//ABS(m_cmdJntPos[7]-curJntPos[7])> m_maxTrackErr OR
//Calculate the deviation of J4 from the zero point
m_instruZeroDeviationJ4:=m_PowerboxZeroPos[1,4] - i_slaveArm.linkSingle[4+3] ;
IF m_instruZeroDeviationJ4>2*PI THEN
	m_instruZeroDeviationJ4:=m_instruZeroDeviationJ4-2*PI;
END_IF

// traj plan
FOR i:=1 TO 5 DO
	m_jntOTG[i].run(m_targetMountPos[i+3],0.0, o_cmdAcc=>m_cmdJntAcc[3+i],o_cmdVel=>m_cmdJntVel[3+i],o_cmdPos=>m_cmdJntPos[i+3]);
END_FOR
END_METHOD

METHOD PUBLIC init : BOOL
VAR_IN_OUT CONSTANT
	i_slaveArm	:FB_SlaveArm;
END_VAR
VAR_IN_OUT 
	r_slaveArmCtrlCmd :ST_SlaveArmCtrlCmds;
END_VAR

VAR
	i : INT;
END_VAR
SUPER^.Init(i_slaveArm,r_slaveArmCtrlCmd);

// check if to hold the command joint position unchanged
checkToHoldLastCmds(i_slaveArm,r_slaveArmCtrlCmd);
FOR i:=1 TO 5 DO
	m_targetMountPos[i+3]:=m_cmdJntPos[i+3];
	m_jntOTG[i].init(m_targetMountPos[i+3], 0,m_instruMountVel, m_instruMountAcc, g_slaveArmCtrlCycleTime);
	m_jointMounted[i]:=FALSE;
END_FOR

m_mountStatus:=0;
// check instrument type to get mount joint index and zero position
IF i_slaveArm.instrument.InstruReadPara.m_Instrutype <> InstruType_UNKNOWM THEN
	m_jointMounted[5]:=TRUE;

END_IF


//Update the IP and port number of the operating arm
i_slaveArm.instrument.InstruReadPara.i_ArmNetId:=GVL_SlaveMotorParameters.g_slaveArmNetID[1];
i_slaveArm.instrument.InstruReadPara.i_JointInstruAddr:=GVL_SlaveMotorParameters.g_slaveJointNetPort[1,4];

m_Error:=FALSE;
m_ErrorID:=0;
END_METHOD

END_FUNCTION_BLOCK

// ---- FBs_SlaveControllers/FB_SlaveCtrlMasterSlave.TcPOU
// Brief: Slave Arm MasterSlave controller
FUNCTION_BLOCK PUBLIC FB_SlaveCtrlMasterSlave EXTENDS FB_SlaveArmCtrlBase
VAR_INPUT
END_VAR
VAR_OUTPUT
END_VAR
VAR
// ################ variables for single joint test ##################
	m_initJntPos :Vec8d;
	m_jntMotionFreq :Vec8d :=[0.1, 0.1, 0.1, 0, 0, 0, 0, 0];
	m_jntMotionRange :Vec8d :=[pi/6, pi/4, 0.1, 0, 0, 0, 0];
	testIdx :INT :=1;
	
//####################################################################

END_VAR

METHOD PROTECTED calcCmdJntPos : BOOL
VAR_INPUT
	motionScale :LREAL;
	masterIdx :INT;
END_VAR

VAR_IN_OUT CONSTANT
	i_slaveArm :FB_SlaveArm;
	i_masterStatus :ST_MasterStatus;
END_VAR
VAR 
	i:INT :=0;
	errThres :LREAL;
END_VAR
// Just for joint controller test
IF testIdx >0 THEN
	m_cmdJntPos[testIdx]:=m_initJntPos[testIdx]+m_jntMotionRange[testIdx]* SIN(2*pi*m_jntMotionFreq[testIdx]*m_timePeriod);
	m_cmdJntVel[testIdx]:=m_jntMotionRange[testIdx]*2*pi*m_jntMotionFreq[testIdx]*COS(2*pi*m_jntMotionFreq[testIdx]*m_timePeriod);
END_IF



FOR i:=1 TO 8 DO 
	IF i=3 THEN
		errThres := 0.01;
	ELSE
		errThres :=5*g_deg2rad;
	END_IF
	
	IF ABS(m_cmdJntPos[i]-i_slaveArm.curJntPos[i])>errThres THEN
		m_isFinished:=TRUE;
	END_IF
	
END_FOR
END_METHOD

// override this function in each exact controller
METHOD PROTECTED calcCmdJntTrq : BOOL
VAR_INPUT
	motionScale :LREAL;
	masterIdx :INT;
END_VAR

VAR_IN_OUT CONSTANT
	i_slaveArm :FB_SlaveArm;
	i_masterStatus :ST_MasterStatus;
END_VAR
VAR 
	nullspaceMat :Mat7d;
	ctrlTrq : Vec7d;
END_VAR
// set joint torque to zero in default
m_cmdJntTrq := g_zeroVec8d;
END_METHOD

METHOD PUBLIC init : BOOL
VAR_IN_OUT CONSTANT
	i_slaveArm	:FB_SlaveArm;
END_VAR
VAR_IN_OUT 
	r_slaveArmCtrlCmd :ST_SlaveArmCtrlCmds;
END_VAR
SUPER^.Init(i_slaveArm,r_slaveArmCtrlCmd);

m_jntOPMode := g_slaveAllPosTrqMode;

m_initJntPos :=i_slaveArm.curJntPos;
END_METHOD

END_FUNCTION_BLOCK

// ---- FBs_SlaveControllers/FB_SlaveCtrlScopeReady.TcPOU
// Brief:Scope Ready
FUNCTION_BLOCK PUBLIC FB_SlaveCtrlScopeReady EXTENDS FB_SlaveArmCtrlBase
VAR_INPUT
END_VAR
VAR_OUTPUT
END_VAR
VAR
END_VAR

METHOD PUBLIC init : BOOL
VAR_IN_OUT CONSTANT
	i_slaveArm	:FB_SlaveArm;
END_VAR
VAR_IN_OUT 
	r_slaveArmCtrlCmd :ST_SlaveArmCtrlCmds;
END_VAR


VAR
	j:INT;
	maxJntErr:LREAL;
	jntCtrlErr:Vec7d;
END_VAR
SUPER^.Init(i_slaveArm,r_slaveArmCtrlCmd);

// check if to hold the command joint position unchanged
checkToHoldLastCmds(i_slaveArm,r_slaveArmCtrlCmd);
END_METHOD

END_FUNCTION_BLOCK

// ---- FBs_SlaveControllers/FB_SlaveCtrlEndoscope.TcPOU
// Brief: Slave Arm Endoscope Control
FUNCTION_BLOCK PUBLIC FB_SlaveCtrlEndoscope EXTENDS FB_SlaveArmCtrlBase
VAR_INPUT
END_VAR
VAR_OUTPUT
END_VAR
VAR
END_VAR

END_FUNCTION_BLOCK

// ---- FBs_SlaveControllers/FB_SlaveCtrlAdjust.TcPOU
// Brief: Slave Arm Adjust
FUNCTION_BLOCK PUBLIC FB_SlaveCtrlAdjust EXTENDS FB_SlaveArmCtrlBase
VAR_INPUT
END_VAR
VAR_OUTPUT
END_VAR
VAR
END_VAR

METHOD PUBLIC init : BOOL
VAR_IN_OUT CONSTANT
	i_slaveArm	:FB_SlaveArm;
END_VAR
VAR_IN_OUT 
	r_slaveArmCtrlCmd :ST_SlaveArmCtrlCmds;
END_VAR
SUPER^.Init(i_slaveArm,r_slaveArmCtrlCmd);

// check if to hold the command joint position unchanged
checkToHoldLastCmds(i_slaveArm,r_slaveArmCtrlCmd);
END_METHOD

END_FUNCTION_BLOCK

// ---- FBs_SlaveControllers/FB_SlaveCtrlGraCali.TcPOU
// Brief: Slave Arm Gravity Calibration
FUNCTION_BLOCK PUBLIC FB_SlaveCtrlGraCali EXTENDS FB_SlaveArmCtrlBase
VAR_INPUT
END_VAR
VAR_OUTPUT
END_VAR
VAR
// cali trajectory
	m_caliMotionSegs :INT :=3;
	m_graCaliTraj:ARRAY [1..3, 1..g_sJntNum] OF LREAL:=
		[-pi/6, -PI/2+pi/6, 0.4, 	0, 0, 0, 0,0,
		 pi/6, 	-PI/2-pi/4, 0.2, 	0, 0, 0, 0,0,
		 -pi/6, -PI/2+pi/6, 0.4, 	0, 0, 0, 0,0];
		 
	m_caliMaxjntVel:Vec8d:=[8(0.02)];
	m_caliMaxjntAcc:Vec8d:=[8(0.5)];
	m_caliMaxjntJerk:Vec8d:=[8(2.0)];
	
	m_caliTrajIdx: INT := 1;
	m_caliPlanner: ARRAY[1..3] OF FB_TrajMoveJ;
	
END_VAR

// override this function in each exact controller
METHOD PROTECTED calcCmdJntPos : BOOL
VAR_INPUT
	motionScale :LREAL;
	masterIdx :INT;
END_VAR

VAR_IN_OUT CONSTANT
	i_slaveArm :FB_SlaveArm;
	i_masterStatus :ST_MasterStatus;
END_VAR

VAR 
	i :INT;
	curJntVel :Vec8d;
END_VAR
// check if planner is ready
IF m_caliPlanner[m_caliTrajIdx].isGene = FALSE THEN
	calcCmdJntPos:=FALSE;
	RETURN;
END_IF

// traj plan
calcCmdJntPos :=m_caliPlanner[m_caliTrajIdx].evaluate(m_timePeriod, jntPos=> m_cmdJntPos, jntVel=>m_cmdJntVel, jntAcc=> m_cmdJntAcc);

// check if to transit to next segment
curJntVel :=i_slaveArm.curJntVel;
IF(m_timePeriod > m_caliPlanner[m_caliTrajIdx].duration  AND vecNorm(curJntVel)<7*GVL_SlaveControlParameters.g_jntStaticVelThres) THEN
	m_caliTrajIdx:=m_caliTrajIdx+1;
	m_timePeriod:=0;
END_IF

// check if to terminated
IF(m_caliTrajIdx > m_caliMotionSegs) THEN
	m_isFinished:=TRUE;
END_IF
END_METHOD

METHOD PUBLIC init : BOOL
VAR_IN_OUT CONSTANT
	i_slaveArm	:FB_SlaveArm;
END_VAR
VAR_IN_OUT 
	r_slaveArmCtrlCmd :ST_SlaveArmCtrlCmds;
END_VAR

VAR
	i,j :INT;
	startJntPos,endJntPos :Vec8d;
END_VAR
SUPER^.Init(i_slaveArm,r_slaveArmCtrlCmd);
m_caliTrajIdx :=1;

// traj plan
// fisrt segment
startJntPos:=i_slaveArm.curJntPos;
FOR j:=1 TO g_sJntNum DO 
endJntPos[j]:=m_graCaliTraj[1,j];
END_FOR
m_caliPlanner[1].init(startJntPos,endJntPos,m_caliMaxjntVel, m_caliMaxJntAcc, m_caliMaxJntJerk);

// other segments
FOR i:=2 TO m_caliMotionSegs DO 
	FOR j:=1 TO g_sJntNum DO 
		startJntPos[j]:=m_graCaliTraj[i-1,j];
		endJntPos[j]:=m_graCaliTraj[i,j];
	END_FOR
	m_caliPlanner[i].init(startJntPos,endJntPos,m_caliMaxjntVel, m_caliMaxJntAcc, m_caliMaxJntJerk);
END_FOR
END_METHOD

END_FUNCTION_BLOCK

// ---- AgiMaths/deg2rad.TcPOU
FUNCTION deg2rad : lreal
VAR_INPUT
	angle_deg:lreal;
END_VAR
VAR
END_VAR

deg2rad:=angle_deg*pi/180;

END_FUNCTION

// ---- FBs_BasicControllers/FBMacroJntControl.TcPOU
// Author: Feijian Ni
// Date: 2023.11.22
FUNCTION_BLOCK FBMacroJntControl
VAR_INPUT
END_VAR
VAR_OUTPUT
END_VAR
VAR
	//TODO: move to GVLs 
	// control paramters
	m_macroJntKp:ARRAY[1..3] OF LREAL:=[1200,10,10];
	m_macroJntKd:ARRAY[1..4] OF LREAL:=[100,1.0,1.0];
	m_macroJntKi:ARRAY[1..4] OF LREAL:=[3000,0,0,0];
	m_macroJntKiLimit:ARRAY[1..4] OF LREAL:=[3(1500.0)];
	m_macroJnttrlLimit:ARRAY[1..4] OF LREAL:=[3(3500.0)];
	m_jntTargetPosLpfCutoffFreq:LREAL:=10;
	m_curJntVelLpfCutoffFreq:LREAL:=30;
	
	// filter for target joint position
	m_cmdPosLpf:ARRAY[1..3] OF FBLowPassFilter;
	
	// filter for current joint velocity
	m_curJntVelLpf:ARRAY[1..3] OF FBLowPassFilter;
	
	// max command joint velocity
	m_maxJntVel:ARRAY[1..3] OF LREAL:=[1.5, 0.1, 0.1];
	
	// arm index for grip control
	m_armIdx:INT;
	
	// final target macro joint position
	m_targetJntPos:ARRAY[1..3] OF LREAL;
	
	// position tracking error
	m_posErr:ARRAY[1..3] OF LREAL;
	
	// max position error for safety check
	m_safetyPosErr:ARRAY[1..3] OF LREAL:=[5.0*pi/180,5.0*pi/180,0.01];
	
	// command macro joint position and veloicty for next cycle
	m_cmdJntPos:ARRAY[1..3] OF LREAL;
	m_cmdJntVel:ARRAY[1..3] OF LREAL;

	// current  macro joint position and veloicty for next cycle
	m_curJntPos:ARRAY[1..3] OF LREAL;
	m_curJntVel:ARRAY[1..3] OF LREAL;
	
	// PID for joint position
	m_jntPIDCtrl:ARRAY[1..3] OF FBPID;
	m_jntCtrlTrq:ARRAY[1..3] OF LREAL;
	
END_VAR

METHOD init : BOOL
VAR_INPUT
	i_armIdx:INT;
END_VAR

VAR
	i,j:INT;
	currentRatioMotor2Jnt:LREAL;
END_VAR
m_armIdx:=i_armIdx;

// get current instrument orientation
m_curJntPos[1]:=Robot_Status.Robot_Current_DH_Joint_Position_M3[m_armIdx].q1;
m_curJntPos[2]:=Robot_Status.Robot_Current_DH_Joint_Position_M3[m_armIdx].q2;
m_curJntPos[3]:=Robot_Status.Robot_Current_DH_Joint_Position_M3[m_armIdx].q3;
FOR i:=1 TO 3  DO 
	m_targetJntPos[i]:=m_curJntPos[i];
	m_cmdJntPos[i]:=m_curJntPos[i];
	m_cmdJntVel[i]:=0;
	m_curJntVel[i]:=0;
END_FOR

// init controller
FOR i:=1 TO 3 DO
	currentRatioMotor2Jnt:=GVL_system_parameters.arm_joint_transmition_efficiency[i-1+Gvl_IO.Joint6]*GVL_system_parameters.arm_joint_torque_constant[i-1+Gvl_IO.Joint6]
							*GVL_system_parameters.transmission_ratio[m_armIdx, i-1+Gvl_IO.Joint6]/1000;
	m_jntPIDCtrl[i].init(GVL_system_parameters.cycle_robot,m_macroJntKp[i],m_macroJntKd[i],m_macroJntKi[i],
		m_macroJntKiLimit[i]* currentRatioMotor2Jnt,	m_macroJnttrlLimit[i]*currentRatioMotor2Jnt);
END_FOR

// init low pass filter
FOR i:=1 TO 3 DO
	m_cmdPosLpf[i].init(i_filterOrd:=1,i_cutoffFreq:=m_jntTargetPosLpfCutoffFreq,i_sampleFreq:=1000);
	m_curJntVelLpf[i].init(i_filterOrd:=1,i_cutoffFreq:=m_curJntVelLpfCutoffFreq,i_sampleFreq:=1000);
END_FOR
END_METHOD

METHOD run : BOOL
VAR_INPUT
	// target joint position in DH model 3
	i_targetJntPos:ARRAY[1..3] OF LREAL;

END_VAR

VAR_OUTPUT
	// motor control current
	o_cmdMotorTrq:ARRAY[1..3] OF LREAL;
END_VAR

VAR
	i: INT;
END_VAR
// fitl target joint position
FOR i:=1 TO 3 DO
	m_targetJntPos[i]:=m_cmdPosLpf[i].run(i_targetJntPos[i]);
END_FOR

// get current joint position
m_curJntPos[1]:=Robot_Status.Robot_Current_DH_Joint_Position_M3[m_armIdx].q1;
m_curJntPos[2]:=Robot_Status.Robot_Current_DH_Joint_Position_M3[m_armIdx].q2;
m_curJntPos[3]:=Robot_Status.Robot_Current_DH_Joint_Position_M3[m_armIdx].q3;

// get current joint velocity
m_curJntVel[1]:=m_curJntVelLpf[1].run(Robot_Status.Robot_Current_Joint_Velocity_V2[m_armIdx,6]);
m_curJntVel[2]:=m_curJntVelLpf[2].run(Robot_Status.Robot_Current_Joint_Velocity_V2[m_armIdx,10]);
m_curJntVel[3]:=m_curJntVelLpf[3].run(Robot_Status.Robot_Current_Joint_Velocity_V2[m_armIdx,11]);

// interpolate command position
FOR i:=1 TO 3 DO
	m_cmdJntVel[i]:=LIMIT(-m_maxJntVel[i],(m_targetJntPos[i]-m_cmdJntPos[i])/GVL_system_parameters.cycle_robot, m_maxJntVel[i]);
	m_cmdJntPos[i]:=m_cmdJntPos[i]+m_cmdJntVel[i]*GVL_system_parameters.cycle_robot;
END_FOR  

// joint position control torque control
FOR i:=1 TO 3 DO
	o_cmdMotorTrq[i]:=0;
	m_posErr[i]:=m_cmdJntPos[i]-m_curJntPos[i];
	m_jntCtrlTrq[i]:=m_jntPIDCtrl[i].run(m_cmdJntPos[i],m_curJntPos[i], m_cmdJntVel[i], m_curJntVel[i]);
END_FOR

// safety check
FOR i:=1 TO 3 DO
	IF ABS(m_posErr[i])>m_safetyPosErr[i] THEN
		run := FALSE;
		RETURN;
	END_IF
END_FOR

// motor control current
o_cmdMotorTrq[1]:=gvl_system_parameters.Joint_Motion_direction[m_armIdx,6]*(m_jntCtrlTrq[1]+Robot_Status.Robot_Joint_Gravity[1].q6);
o_cmdMotorTrq[2]:=gvl_system_parameters.Joint_Motion_direction[m_armIdx,10]*(m_jntCtrlTrq[2]+Robot_Status.Robot_Joint_Gravity[1].q10);
o_cmdMotorTrq[3]:=gvl_system_parameters.Joint_Motion_direction[m_armIdx,11]*(m_jntCtrlTrq[3]+Robot_Status.Robot_Joint_Gravity[1].q11);
run := TRUE;
END_METHOD

END_FUNCTION_BLOCK

// ---- FBs_RobotDynamics/FB_SlaveGravity.TcPOU
FUNCTION_BLOCK FB_SlaveGravity
VAR_INPUT
END_VAR
VAR_OUTPUT
END_VAR
VAR
	// arm index
	m_armIdx :INT;
	
	(*graParam=[ 2.7244*m3 + 2.7244*m4 + 2.7244*m5 + 2.7244*m6 + 9.8*mx2 + 9.8*mx9,
            	9.8*my2 + 9.8*my9,
			 	3.577*m4 + 3.577*m5 + 3.577*m6 + 0.49*m9 + 9.8*mx3 + 9.8*mx8
           		1.5827*m4 + 1.5827*m5 + 1.5827*m6 + 9.8*my3 + 9.8*my8 + 9.8*mz4
            	mz5-my4,	my5+mz6,  	mx4,   	mx5, 	mx6,   	my6
            	preF2,   k2,   preF3,    k3,    preF5   k5]*)
	m_gravityParam :ARRAY[1..16] OF REAL;
	// spring2 [L0, b1, b2, l1, r0]
	m_spring2Param :ARRAY[1..5] OF LREAL;
	// spring3 [L0, b1, b2, l1, r0,d]
	m_spring3Param :ARRAY[1..6] OF LREAL;
	// spring5 [L0, s1, L1, r0, beta]
	m_spring5Param :ARRAY[1..5] OF LREAL;
END_VAR

METHOD PUBLIC init : BOOL
VAR_INPUT
	i_armIdx :INT;
END_VAR
VAR
	i:INT;
END_VAR
m_armIdx:=i_armIdx;
END_METHOD

METHOD PUBLIC run : BOOL
VAR_IN_OUT CONSTANT
	// slave arm joint position
	i_jntPos :vec8d;
	
	// set up distal end frame
	i_setArmFrame : ST_Frame;
END_VAR
VAR_IN_OUT
	r_gravity :Vec3d;
END_VAR
VAR


END_VAR
r_gravity := g_zeroVec3d;
END_METHOD

END_FUNCTION_BLOCK

// ---- FBs_Robots/FB_SetupArm.TcPOU
FUNCTION_BLOCK FB_SetupArm
VAR_INPUT
END_VAR
VAR_OUTPUT
END_VAR
VAR
	// arm index, from 1 to 4
	m_armIdx: INT;
	
	// joints
	m_joints :ARRAY[1..g_sJntNum] OF FB_SetupJoint;
	
	// IO
	m_manualAdjustIO AT%I* :SINT;
	m_manualAdjustOnFlag :BOOL;
	m_autoAdjustIO AT%I* :SINT;
	m_autoAdjustDir :INT; // -1, 0, 1;
	
	// arm cartesian data, defined in cart origin
	m_curCartPose	:ST_Frame;
	
	// cartesion position of remote center
	m_rcPos :Vec3d;	
	
	// arm joint data
	m_curMotorPos :Vec5d;
	m_curLinkPos :Vec5d;
	m_curJntPos :Vec5d;
	m_curJntVel :Vec5d;
	m_curJntTrq :Vec5d;
	m_cmdJntTrq :Vec5d;
	m_rawJntCurrent :Vec5d;
	m_filtJntCurrent :Vec5d;
	m_cmdJntCurrent : Vec5d;
		
	// arm gravity
	m_jntGravity : Vec5d:=g_zeroVec5d;
	
	
END_VAR

PROPERTY armIdx : int
GET
armIdx:=m_armIdx;
END_GET
END_PROPERTY

// check auto adjust direction
METHOD autoAdjustDetect : INT
VAR_INPUT
END_VAR
// TODO
END_METHOD

PROPERTY autoAdjustDir : INT
GET
autoAdjustDir := m_autoAdjustDir;
END_GET
END_PROPERTY

METHOD checkIO : BOOL
VAR_INPUT
END_VAR
// check manual and auto adjust button
m_manualAdjustOnFlag := manualAdjustDetect();
m_autoAdjustDir :=autoAdjustDetect();
END_METHOD

PROPERTY cmdJntCurrent : REFERENCE TO  Vec5d
GET
cmdJntCurrent ref= m_cmdJntCurrent;
END_GET
END_PROPERTY

PROPERTY curCartPose : REFERENCE TO ST_Frame
GET
curCartPose ref=m_curCartPose;
END_GET
END_PROPERTY

PROPERTY curJntPos : REFERENCE TO Vec5d
GET
curJntPos ref=m_curJntPos;
END_GET
END_PROPERTY

PROPERTY curJntTrq : REFERENCE TO Vec5d
GET
curJntTrq ref=m_curJntTrq;
END_GET
END_PROPERTY

PROPERTY curJntVel :REFERENCE TO Vec5d
GET
curJntVel ref=m_curJntVel;
END_GET
END_PROPERTY

PROPERTY curLinkPos :REFERENCE TO Vec5d
GET
curLinkPos ref=m_curLinkPos;
END_GET
END_PROPERTY

PROPERTY curMotorPos : REFERENCE TO  Vec5d
GET
curMotorPos ref=m_curMotorPos;
END_GET
END_PROPERTY

METHOD PUBLIC enable : BOOL
VAR_IN_OUT CONSTANT
	i_jntIdx :Vec5i;
END_VAR
VAR
	i :INT ;
END_VAR
FOR i:=1 TO g_setupJntNum DO
	IF 1= i_jntIdx[i] THEN
		m_joints[i].enable();
	ELSE
		m_joints[i].disable();
	END_IF
END_FOR
END_METHOD

PROPERTY filtJntCurrent :REFERENCE TO Vec5d
GET
filtJntCurrent ref= m_filtJntCurrent;
END_GET
END_PROPERTY

// compute cartesion pose in cart origin
METHOD PROTECTED forwardKinematic : BOOL
VAR_IN_OUT CONSTANT
	i_jntPos :Vec5d;
END_VAR
VAR_IN_OUT
	r_cartPose :ST_Frame;
	
	// position of remote center
	r_rcPos :Vec3d;
END_VAR
VAR
	a2,d4,d6:LREAL; //DH parameters
	
	Radius,Angle,R1,q:LREAL; //Disk structure parameters
	x,y,z:LREAL;
	basePosMatrix:ARRAY[1..4,1..4] OF LREAL;//transform from origin to C0
	
	T_50:ARRAY[1..4,1..4] OF LREAL; //transform from C0 to C5
	F5:ARRAY[1..4,1..4] OF LREAL; //transform from origin to C5
	q1,q2,q3,q4,q5:LREAL;	
	c14,s14,c5,s5,s1,c1:LREAL;
	
	fixPointTransform:ARRAY[1..4,1..4] OF LREAL; //transform from C5 to fixed point
	fixPointMatrix:ARRAY[1..4,1..4] OF LREAL;
END_VAR
//TODO


//****************input:five joint position of SetupArm********************//
q1:=i_jntPos[1]; q2:=i_jntPos[2]; q3:=i_jntPos[3]; q4:=i_jntPos[4]; q5:=i_jntPos[5];




//**********************DH parameters*************************//
IF (m_armIdx=1) THEN
	a2:=0.019; d4:=0.3545;
	
ELSIF (m_armIdx=2) THEN
	a2:=0.136; d4:=0.3545;
	
ELSIF (m_armIdx=3) THEN	
	a2:=0.136; d4:=0.5205;
	
ELSIF (m_armIdx=4) THEN	
	a2:=0.1825; d4:=0.5205;
END_IF
d6:=0.6387229+0.1659;



//********************transform form origin to C0***********************//
Radius:=0.170; Angle:=deg2rad(60);
R1:=Radius;  q:=Angle;
IF (m_armIdx=1) THEN
	x:=-R1; y:=0; z:=0;
	
ELSIF (m_armIdx=2) THEN
	x:=-R1*COS(q); y:=-R1*SIN(q); z:=0;
	
ELSIF (m_armIdx=3) THEN	
	x:=R1*COS(q); y:=-R1*SIN(q); z:=0;
	
ELSIF (m_armIdx=4) THEN	
	x:=R1; y:=0; z:=0;
END_IF

basePosMatrix[1,1]:=0;
basePosMatrix[2,1]:=1;
basePosMatrix[3,1]:=0;
basePosMatrix[4,1]:=0;

basePosMatrix[1,2]:=-1;
basePosMatrix[2,2]:=0;
basePosMatrix[3,2]:=0;
basePosMatrix[4,2]:=0;

basePosMatrix[1,3]:=0;
basePosMatrix[2,3]:=0;
basePosMatrix[3,3]:=1;
basePosMatrix[4,3]:=0;

basePosMatrix[1,4]:=x;
basePosMatrix[2,4]:=y;
basePosMatrix[3,4]:=z;
basePosMatrix[4,4]:=1;




//***************output1:C5 posture relative to origin(other than C0)*************//
c14:=COS(q1+q4); s14:=SIN(q1+q4); 
c5:=COS(q5); s5:=SIN(q5);
c1:=COS(q1); s1:=SIN(q1);

T_50[1,1]:=c14*c5; 
T_50[2,1]:=s14*c5; 
T_50[3,1]:=-s5; 
T_50[4,1]:=0;

T_50[1,2]:=-c14*s5;
T_50[2,2]:=-s14*s5; 
T_50[3,2]:=-c5; 
T_50[4,2]:=0;

T_50[1,3]:=-s14;
T_50[2,3]:=c14;
T_50[3,3]:=0;
T_50[4,3]:=0;

T_50[1,4]:=a2*c1 + q2*s1;
T_50[2,4]:=a2*s1 - q2*c1;
T_50[3,4]:=d4 + q3;
T_50[4,4]:=1;

matMultiply(basePosMatrix,T_50,F5);
r_cartPose.m_pos[1]:=F5[1,4]; r_cartPose.m_pos[2]:=F5[2,4]; r_cartPose.m_pos[3]:=F5[3,4];

r_cartPose.m_rot[1,1]:=F5[1,1];  r_cartPose.m_rot[1,2]:=F5[1,2];  r_cartPose.m_rot[1,3]:=F5[1,3];
r_cartPose.m_rot[2,1]:=F5[2,1];  r_cartPose.m_rot[2,2]:=F5[2,2];  r_cartPose.m_rot[2,3]:=F5[2,3];
r_cartPose.m_rot[3,1]:=F5[3,1];  r_cartPose.m_rot[3,2]:=F5[3,2];  r_cartPose.m_rot[3,3]:=F5[3,3];




//********************output2:remote center position************************//
fixPointTransform[1,1]:=1;  fixPointTransform[2,2]:=1;  fixPointTransform[3,3]:=1;  fixPointTransform[4,4]:=1;  
fixPointTransform[2,4]:=-d6;  
matMultiply(F5,fixPointTransform,fixPointMatrix);
r_rcPos[1]:=fixPointMatrix[1,4];  r_rcPos[2]:=fixPointMatrix[2,4];  r_rcPos[3]:=fixPointMatrix[3,4];
END_METHOD

METHOD PUBLIC init : BOOL
VAR_INPUT
	i_armIdx:INT;
END_VAR
VAR 
	i :INT ;
END_VAR
// arm statues init
m_armIdx:=i_armIdx;

// joint init
FOR i:=1 TO g_setupJntNum DO
	m_joints[i].init(m_armIdx, i);
END_FOR

// init joint encoder and position calculation
initJntPos();

// compute current status
updateStatus();
END_METHOD

METHOD initJntPos : BOOL
VAR_INPUT
END_VAR
VAR
	i:INT ;
END_VAR
// joint init
FOR i:=1 TO g_setupJntNum DO
	m_joints[i].initJntPos();
END_FOR
END_METHOD

// check if instrument is on
METHOD instruDetect : BOOL
VAR_INPUT
END_VAR
//TODO
END_METHOD

METHOD PUBLIC isEnabled : BOOL
VAR_IN_OUT CONSTANT
	i_jntIdx :Vec5i;
END_VAR
VAR
	i :INT ;
END_VAR
isEnabled := TRUE;
FOR i:=1 TO g_setupJntNum DO
	IF 1= i_jntIdx[i] THEN
		isEnabled :=  (m_joints[i].isEnabled() AND isEnabled);
	END_IF
END_FOR
END_METHOD

PROPERTY jntGravity :REFERENCE TO Vec5d
GET
jntGravity ref=m_jntGravity;
END_GET
END_PROPERTY

// check if adjust button is pressed
METHOD manualAdjustDetect : BOOL
VAR_INPUT
END_VAR
// TODO
END_METHOD

PROPERTY manualAdjustOn : bool
GET
manualAdjustOn := m_manualAdjustOnFlag;
END_GET
END_PROPERTY

PROPERTY rawJntCurrent :REFERENCE TO Vec5d
GET
rawJntCurrent ref=m_rawJntCurrent;
END_GET
END_PROPERTY

PROPERTY rcPos :REFERENCE to Vec3d
GET
rcPos REF= m_rcPos;
END_GET
END_PROPERTY

// update joints control command
METHOD PUBLIC updateCmds : BOOL
VAR_IN_OUT CONSTANT
	i_armCtrlCmd : ST_SetupArmCtrlCmds;
END_VAR
VAR
	i:INT;
END_VAR
m_cmdJntTrq:=i_armCtrlCmd.m_cmdJntTrq;

// enable/disable joints
enable(i_armCtrlCmd.m_jntEnableFlag);

// position/torque control
FOR i:=1 TO g_setupJntNum DO 
	IF i_armCtrlCmd.m_jntOPMode[i]=DriverOPMode_Trq THEN
		// gravity feedforward
		m_cmdJntTrq[i]:=m_cmdJntTrq[i]+m_jntGravity[i];
		m_joints[i].updateCmds(DriverOPMode_Trq,i_armCtrlCmd.m_cmdJntPos[i],m_cmdJntTrq[i]);
	ELSE
		m_cmdJntTrq[i]:=0;
		m_joints[i].updateCmds(DriverOPMode_Pos,i_armCtrlCmd.m_cmdJntPos[i],m_cmdJntTrq[i]);
	END_IF
	
END_FOR
END_METHOD

METHOD PUBLIC updateDyna : BOOL
VAR_IN_out constant
	i_jnt3Gravity :LREAL;
	i_jnt5Gravity :LREAL;
END_VAR
m_jntGravity[3]:=i_jnt3Gravity;
m_jntGravity[5]:=i_jnt5Gravity;
END_METHOD

// update arm status, including kinematic and dynamic
METHOD PUBLIC updateStatus : BOOL
VAR_INPUT
END_VAR
VAR 
	i,j:INT;
END_VAR
// update joint data
FOR i:=1 TO g_setupJntNum DO
	m_joints[i].updateStatus();
END_FOR

// check adjust button
checkIO();

// get joint data
FOR i:=1 TO g_setupJntNum DO
	m_curMotorPos[i]:=m_joints[i].motorPos;
	m_curLinkPos[i]:=m_joints[i].linkPos;
	m_curJntPos[i]:=m_joints[i].jntPos;
	m_curJntVel[i]:=m_joints[i].jntVel;
	m_curJntTrq[i]:=m_joints[i].jntTrq;
	m_rawJntCurrent[i]:=m_joints[i].rawCurrent;
	m_filtJntCurrent[i]:=m_joints[i].filtCurrent;
	m_cmdJntCurrent[i]:=m_joints[i].cmdCurrent;
END_FOR 

// cartesion pose
forwardKinematic(m_curJntPos,m_curCartPose,m_rcPos);
END_METHOD

END_FUNCTION_BLOCK

// ---- FBs_Robots/FB_SetupJoint.TcPOU
FUNCTION_BLOCK FB_SetupJoint EXTENDS FB_JointBase
VAR_INPUT
END_VAR
VAR_OUTPUT
END_VAR
VAR
END_VAR

METHOD init : BOOL
VAR_INPUT
	i_armIdx :INT;
	i_jntIdx :INT;
	i_controlCycleTime :LREAL;
END_VAR
m_cycleTime := i_controlCycleTime;

// hardware parameters
m_motorEncoderRes :=GVL_SetupMotorParameters.g_incEncoderRes[i_jntIdx];
m_linkEncoderRes :=GVL_SetupMotorParameters.g_absEncoderRes[i_jntIdx];
m_motorReduction :=GVL_SetupMotorParameters.g_motorReduction[i_jntIdx];
m_linkEncoderReduction :=GVL_SetupMotorParameters.g_absEncoderReduction[i_jntIdx];
m_trqConst :=GVL_SetupMotorParameters.g_motorTrqConst[i_jntIdx];
m_maxCurrent :=GVL_SetupMotorParameters.g_motorMaxCurrent[i_jntIdx];
m_motorDir :=GVL_SetupMotorParameters.g_motorDir[i_jntIdx];								
m_linkEncoderDir :=GVL_SetupMotorParameters.g_asbEncoderDir[i_jntIdx];
m_minJntPos	:=GVL_SetupMotorParameters.g_minJntPos[i_jntIdx];
m_maxJntPos	:=GVL_SetupMotorParameters.g_maxJntPos[i_jntIdx];

//link encoder calibartion data
m_minLinkEncoder :=GVL_SetupJointEncoderCaliData.g_minLinkEncoder[i_armIdx, i_jntIdx] - m_linkEncoderDir*GVL_SlaveJointEncoderCaliData.g_linkEncLimitBuffer; // expand limit
m_maxLinkEncoder :=GVL_SetupJointEncoderCaliData.g_maxLinkEncoder[i_armIdx, i_jntIdx] + m_linkEncoderDir*GVL_SlaveJointEncoderCaliData.g_linkEncLimitBuffer; // expand limit
m_caliLinkEncoder :=GVL_SetupJointEncoderCaliData.g_caliLinkEncoder[i_armIdx, i_jntIdx];
m_linkEncCaliJntPos :=GVL_SetupJointEncoderCaliData.g_linkEncCaliJntPos[i_jntIdx];
m_linkEncZeroCross :=GVL_SetupJointEncoderCaliData.g_linkEncZeroCross[i_armIdx, i_jntIdx];
m_multiCycles :=GVL_SetupJointEncoderCaliData.g_multipleCyclesJoint[i_armIdx,i_jntIdx];

// convert cali link encoder if joint cross zero
IF 1=m_linkEncZeroCross THEN
	IF 1=m_linkEncoderDir AND m_caliLinkEncoder < m_minLinkEncoder THEN
		m_caliLinkEncoder := GVL_SetupJointEncoderCaliData.g_caliLinkEncoder[i_armIdx, i_jntIdx] + m_linkEncoderRes;
	ELSIF -1=m_linkEncoderDir AND m_caliLinkEncoder < m_maxLinkEncoder THEN
		m_caliLinkEncoder := GVL_SetupJointEncoderCaliData.g_caliLinkEncoder[i_armIdx, i_jntIdx] + m_linkEncoderRes;
	END_IF
END_IF

// macro data
m_trq2CurrentRatio:=m_motorDir * 1000.0/(m_trqConst*m_motorReduction);
m_current2TrqRatio:=m_motorDir * (m_trqConst*m_motorReduction)/1000.0;
m_linkEnc2PosRatio := 2*PI*m_linkEncoderDir/(m_linkEncoderReduction*m_linkEncoderRes);
m_motorEnc2PosRatio := 2*PI * m_motorDir/(m_motorReduction * m_motorEncoderRes);

// motor data init
m_curJntVel:=0;
m_curJntTrq :=0;
m_rawCurrent :=0;
m_filtCurrent :=0;
m_cmdJntVel :=0.0;
m_cmdJntTrq :=0.0;
m_cmdCurrent := 0.0;

// filter init
m_jntVelLpf.init(1, GVL_SetupControlParameters.g_curJntVelLpfCutoffFreq, g_setupArmCtrlFreq);
m_cmdTrqLpf.init(1, GVL_SetupControlParameters.g_cmdJntTrqLpfCutoffFreq, g_setupArmCtrlFreq);
m_curTrqLpf.init(1, GVL_SetupControlParameters.g_curJntTrqLpfCutoffFreq, g_setupArmCtrlFreq);

// driver init value
m_motorOutputs.m_controlWord:=DriverCtrlWord_INIT;
m_motorOutputs.m_opMode:=INT_TO_SINT(DriverOPMode_Pos);
m_motorOutputs.m_cmdCurrent:=0;
m_motorOutputs.m_cmdMotorEncoder:=m_motorInputs.m_motorEncoder;
END_METHOD

END_FUNCTION_BLOCK

// ---- FBs_Robots/FB_SetupRobot.TcPOU
FUNCTION_BLOCK FB_SetupRobot
VAR_INPUT
END_VAR
VAR_OUTPUT
END_VAR
VAR
	// setup arms, responsible for arm kinematic and control
	m_setupArms :ARRAY[1..g_sArmNum] OF FB_SetupArm;
	
	// arm state
	m_setupArmState:ARRAY[1..g_sArmNum] OF E_setupArmState:=[4(E_setupArmState.SetupArmState_Init)];
	m_lastSetupArmState:ARRAY[1..g_sArmNum] OF E_setupArmState:=[4(E_setupArmState.SetupArmState_Init)];
	m_nextSetupArmState:ARRAY[1..g_sArmNum] OF E_setupArmState:=[4(E_setupArmState.SetupArmState_Init)];
	
	// all arm controller instance 
	m_armCtrlFactory :ARRAY[1..g_sArmNum,1..SetupArmState_totalNum] OF I_SetupArmCtrl;
	m_armInit :ARRAY[1..g_sArmNum] OF FB_SetupCtrlInit;
	m_armError :ARRAY[1..g_sArmNum] OF FB_SetupCtrlError;
	m_armSelfCheck :ARRAY[1..g_sArmNum] OF FB_SetupCtrlSelfCheck;
	m_armHold :ARRAY[1..g_sArmNum] OF FB_SetupCtrlHold;
	m_armManualAdjust :ARRAY[1..g_sArmNum] OF FB_SetupCtrlManualAdjust;
	m_armAutoAdjust :ARRAY[1..g_sArmNum] OF FB_SetupCtrlAutoAdjust;
	m_armPackage :ARRAY[1..g_sArmNum] OF FB_SetupCtrlPackage;
	m_armCart :ARRAY[1..g_sArmNum] OF FB_SetupCtrlCart;
	m_armGraCali :ARRAY[1..g_sArmNum] OF FB_SetupCtrlGraCali;
	
	
	// arm controller interface
	m_armCtrl :ARRAY[1..g_sArmNum] OF I_SetupArmCtrl;
	m_armCtrlCmds :ARRAY[1..g_sArmNum] OF ST_SetupArmCtrlCmds;

END_VAR

METHOD PUBLIC getStatus : BOOL
VAR_IN_OUT
	// slave robot information, including arm status and cartesian data
	r_setupStatus :ST_SetupStatus;
	
	// slave robot joint data
	r_setupJointsData :ST_SetupJointData;
	
END_VAR

VAR
	i:INT;
END_VAR
r_setupStatus.m_armState:=m_setupArmState;

// TODO: project cartesion data to monitor coordinate
FOR i:=1 TO g_sArmNum DO
	
	// cartesion
	r_setupStatus.m_curEndPose[i]:=m_setupArms[i].curCartPose;
	r_setupStatus.m_rcPos[i]:=m_setupArms[i].rcPos;
	
	// joint
	r_setupJointsData.m_curMotorPos[i]:=m_setupArms[i].curMotorPos;
	r_setupJointsData.m_curLinkPos[i]:=m_setupArms[i].curLinkPos;
	r_setupJointsData.m_curJntPos[i]:=m_setupArms[i].curJntPos;
	r_setupJointsData.m_curJntVel[i]:=m_setupArms[i].curJntVel;
	r_setupJointsData.m_curJntTrq[i]:=m_setupArms[i].curJntTrq;
	
	// command info
	// joint info
	r_setupJointsData.m_cmdJntPos[i]:=m_armCtrlCmds[i].m_cmdJntPos;
	r_setupJointsData.m_cmdJntVel[i]:=m_armCtrlCmds[i].m_cmdJntVel;
	r_setupJointsData.m_cmdJntTrq[i]:=m_armCtrlCmds[i].m_cmdJntTrq;
	
END_FOR
END_METHOD

METHOD PUBLIC Init : BOOL
VAR_INPUT
END_VAR
VAR
	i:INT;
END_VAR
FOR i:=1 TO g_sArmNum DO
	// arm init
	m_setupArms[i].Init(i);
	m_setupArmState[i]:=SlaveArmState_Init;
	m_lastSetupArmState[i]:=SlaveArmState_Init;
	m_nextSetupArmState[i]:=SlaveArmState_Init;
	
	// command init
	m_armCtrlCmds[i].m_jntEnableFlag := g_zeroVec5i;
	m_armCtrlCmds[i].m_jntOPMode := g_setupAllPosMode;
	m_armCtrlCmds[i].m_cmdJntPos := m_setupArms[i].curJntPos;
	m_armCtrlCmds[i].m_cmdJntVel := g_zeroVec5d;
	m_armCtrlCmds[i].m_cmdJntAcc := g_zeroVec5d;
	m_armCtrlCmds[i].m_cmdJntTrq := g_zeroVec5d;
	
	// generate controller factory
	m_armCtrlFactory[i,SetupArmState_Error] := m_armError[i];
	m_armCtrlFactory[i,SetupArmState_Init] := m_armInit[i];
	m_armCtrlFactory[i,SetupArmState_SelfCheck] := m_armSelfCheck[i];
	m_armCtrlFactory[i,SetupArmState_Hold] := m_armHold[i];
	m_armCtrlFactory[i,SetupArmState_ManulAdjust] := m_armManualAdjust[i];
	m_armCtrlFactory[i,SetupArmState_AutoAdjust] := m_armAutoAdjust[i];
	m_armCtrlFactory[i,SetupArmState_Package] := m_armPackage[i];
	m_armCtrlFactory[i,SetupArmState_Cart] := m_armCart[i];
	m_armCtrlFactory[i,SetupArmState_GravityCali] := m_armGraCali[i];
	
	// assign controller
	m_armCtrl[i]:=m_armCtrlFactory[i,m_setupArmState[i]];
	m_armCtrl[i].Init(m_setupArms[i],m_armCtrlCmds[i]);
END_FOR
END_METHOD

METHOD PUBLIC run : BOOL
VAR_IN_OUT CONSTANT
	i_setupInputDataPool:ST_SetupInputDataPool;
END_VAR
VAR
	i:INT;
END_VAR
// state machine transition
stateMachine(i_setupInputDataPool);

FOR i:=1 TO g_sArmNum DO
	// update dynamic data
	m_setupArms[i].updateDyna(i_setupInputDataPool.m_setupJnt3Gravity, i_setupInputDataPool.m_setupJnt5Gravity);
								
	// update slave arm kinematics
	m_setupArms[i].updateStatus();
	
	// null ptr check
	IF 0 = m_armCtrl[i] THEN
		EXIT;
	END_IF
	
	// run controller
	m_armCtrl[i].run(m_setupArms[i],m_armCtrlCmds[i]);

	// update commands to drivers
	m_setupArms[i].updateCmds(m_armCtrlCmds[i]);

END_FOR
END_METHOD

// state machine check and transit 
METHOD PROTECTED stateMachine : BOOL
VAR_IN_OUT CONSTANT
		i_setupInputDataPool:ST_SetupInputDataPool;
END_VAR
VAR
	i:INT;
END_VAR
FOR i:=1 TO g_sArmNum DO
	// State machine transit 
	CASE m_setupArmState[i] OF
		// init
		SetupArmState_Init:
			IF m_armCtrl[i].isFinished  THEN
				m_nextSetupArmState[i]:=SetupArmState_SelfCheck;
			END_IF

		//self check
		SetupArmState_SelfCheck:
			IF m_armCtrl[i].isFinished  THEN
				m_nextSetupArmState[i]:=SetupArmState_Hold;
			END_IF
		
		//hold
		SetupArmState_Hold:
			IF m_setupArms[i].manualAdjustOn THEN
				m_nextSetupArmState[i]:=SetupArmState_ManulAdjust;
			ELSIF m_setupArms[i].autoAdjustDir<>0 THEN
				m_nextSetupArmState[i]:=SetupArmState_AutoAdjust;
			END_IF
			
(*		
		//package
		SetupArmState_Package:
		
		//cart
		SetupArmState_Cart:
		
		//gravity calibration
		SetupArmState_GravityCali:
		
*)
	END_CASE
	
	// Controller transit
	IF m_nextSetupArmState[i]<> m_setupArmState[i] THEN
		// reset current controller
		m_armCtrl[i].reset();
		
		// transit to new controller
		m_lastSetupArmState[i]:=m_setupArmState[i];
		m_setupArmState[i]:=m_nextSetupArmState[i];
		m_armCtrl[i]:=m_armCtrlFactory[i,m_setupArmState[i]];
		
		// init next controller
		m_armCtrl[i].Init(m_setupArms[i],m_armCtrlCmds[i]);
		m_setupArms[i].updateCmds(m_armCtrlCmds[i]);
	END_IF
END_FOR
END_METHOD

END_FUNCTION_BLOCK

// ---- FBs_SetupControllers/FB_SetupCtrlSelfCheck.TcPOU
// Brief: Setup Arm Self-check
FUNCTION_BLOCK PUBLIC FB_SetupCtrlSelfCheck EXTENDS FB_SetupArmCtrlBase
VAR_INPUT
END_VAR
VAR_OUTPUT
END_VAR
VAR

	
END_VAR

METHOD PUBLIC init : BOOL
VAR_IN_OUT CONSTANT
	i_setupArm	:FB_SetupArm;
END_VAR
VAR_IN_OUT 
	r_setupArmCtrlCmd :ST_SetupArmCtrlCmds;
END_VAR
SUPER^.Init(i_setupArm,r_setupArmCtrlCmd);
END_METHOD

END_FUNCTION_BLOCK

// ---- FBs_SetupControllers/FB_SetupCtrlHold.TcPOU
// Brief: Setup Arm Init
FUNCTION_BLOCK PUBLIC FB_SetupCtrlHold EXTENDS FB_SetupArmCtrlBase
VAR_INPUT
END_VAR
VAR_OUTPUT
END_VAR
VAR
	m_initState :INT :=0;
END_VAR

END_FUNCTION_BLOCK

// ---- FBs_SetupControllers/FB_SetupCtrlPackage.TcPOU
// Brief: Setup Arm Move to Package Posture
FUNCTION_BLOCK PUBLIC FB_SetupCtrlPackage EXTENDS FB_SetupArmCtrlBase
VAR_INPUT
END_VAR
VAR_OUTPUT
END_VAR
VAR
END_VAR

METHOD PUBLIC init : BOOL
VAR_IN_OUT CONSTANT
	i_setupArm	:FB_SetupArm;
END_VAR
VAR_IN_OUT 
	r_setupArmCtrlCmd :ST_SetupArmCtrlCmds;
END_VAR
SUPER^.Init(i_setupArm,r_setupArmCtrlCmd);
END_METHOD

END_FUNCTION_BLOCK

// ---- FBs_SetupControllers/FB_SetupCtrlCart.TcPOU
// Brief: setup Arm Cart Control
FUNCTION_BLOCK PUBLIC FB_SetupCtrlCart EXTENDS FB_SetupArmCtrlBase
VAR_INPUT
END_VAR
VAR_OUTPUT
END_VAR
VAR
END_VAR

END_FUNCTION_BLOCK

// ---- FBs_SetupControllers/FB_SetupCtrlGraCali.TcPOU
// Brief: setup arm gravity calibration
// For trajectory synchronizaiton, the planner generate a trajecotry for setup joint3/5 and slave joint 1-3, but only former used here 
FUNCTION_BLOCK PUBLIC FB_SetupCtrlGraCali EXTENDS FB_SetupArmCtrlBase
VAR_INPUT
END_VAR
VAR_OUTPUT
END_VAR
VAR
// cali trajectory
	m_caliMotionSegs :INT :=3;
	m_graCaliTraj:ARRAY [1..3, 1..5] OF LREAL:=
		[0,	0,	0.1,	0,	pi/2,
		 0,	0,	0.2,	0,	pi/2+pi/4,
		 0,	0,	0.1,	0,	pi/2-pi/4];
		 
	m_caliMaxjntVel:Vec5d:=[5(0.02)];
	m_caliMaxjntAcc:Vec5d:=[5(0.5)];
	m_caliMaxjntJerk:Vec5d:=[5(2.0)];
	
	m_caliTrajIdx: INT := 1;
	m_caliPlanner: ARRAY[1..3] OF FB_setupTrajMoveJ;
	
END_VAR

// override this function in each exact controller
METHOD PROTECTED calcCmdJntPos : BOOL
VAR_IN_OUT CONSTANT
	i_setupArm	:FB_SetupArm;
END_VAR


VAR 
	i :INT;
	curJntVel :Vec5d;
END_VAR
// check if planner is ready
IF m_caliPlanner[m_caliTrajIdx].isGene = FALSE THEN
	calcCmdJntPos:=FALSE;
	RETURN;
END_IF

// traj plan
calcCmdJntPos :=m_caliPlanner[m_caliTrajIdx].evaluate(m_timePeriod, jntPos=> m_cmdJntPos, jntVel=>m_cmdJntVel, jntAcc=> m_cmdJntAcc);

// check if to transit to next segment
curJntVel :=i_setupArm.curJntVel;
IF(m_timePeriod > m_caliPlanner[m_caliTrajIdx].duration  AND vecNorm(curJntVel)<5*GVL_SlaveControlParameters.g_jntStaticVelThres) THEN
	m_caliTrajIdx:=m_caliTrajIdx+1;
	m_timePeriod:=0;
END_IF

// check if to terminated
IF(m_caliTrajIdx > m_caliMotionSegs) THEN
	m_isFinished:=TRUE;
END_IF
END_METHOD

METHOD PUBLIC init : BOOL
VAR_IN_OUT CONSTANT
	i_setupArm	:FB_SetupArm;
END_VAR
VAR_IN_OUT 
	r_setupArmCtrlCmd :ST_SetupArmCtrlCmds;
END_VAR

VAR
	i,j :INT;
	startJntPos,endJntPos :Vec5d;
END_VAR
SUPER^.Init(i_setupArm,r_setupArmCtrlCmd);
m_caliTrajIdx :=1;

// traj plan
// fisrt segment
startJntPos:=i_setupArm.curJntPos;
FOR j:=1 TO g_setupJntNum DO 
endJntPos[j]:=m_graCaliTraj[1,j];
END_FOR
m_caliPlanner[1].init(startJntPos,endJntPos,m_caliMaxjntVel, m_caliMaxJntAcc, m_caliMaxJntJerk);

// other segments
FOR i:=2 TO m_caliMotionSegs DO 
	FOR j:=1 TO g_setupJntNum DO 
		startJntPos[j]:=m_graCaliTraj[i-1,j];
		endJntPos[j]:=m_graCaliTraj[i,j];
	END_FOR
	m_caliPlanner[i].init(startJntPos,endJntPos,m_caliMaxjntVel, m_caliMaxJntAcc, m_caliMaxJntJerk);
END_FOR
END_METHOD

END_FUNCTION_BLOCK

// ---- FBs_TrajectoryPlanning/FB_setupTrajMoveJ.TcPOU
FUNCTION_BLOCK FB_setupTrajMoveJ EXTENDS FB_TrajBase
VAR_OUTPUT
END_VAR
VAR
	// move vector in joint space
	m_startPos:Vec5d;
	m_targetPos:Vec5d;
	m_moveDir : Vec5d;
	m_moveDistance :LREAL;
	
	// doubleS planning for move distance
	m_doubleS :FB_BasicDoubleS;
END_VAR

METHOD evaluate : BOOL
VAR_INPUT
	t :LREAL;
END_VAR

VAR_OUTPUT
	jntPos,jntVel, jntAcc :vec5d;
END_VAR
VAR
	q,q_dot,q_ddot :LREAL;
	moveRange :Vec5d;
END_VAR
evaluate:=m_doubleS.evaluate(t,q=>q,q_dot=>q_dot, q_ddot=>q_dot);
IF evaluate =FALSE THEN
	RETURN;
END_IF

vecMultiNum(m_moveDir,q, moveRange);
vecAdd(moveRange, m_startPos,jntPos);
vecMultiNum(m_moveDir,q_dot, jntVel);
vecMultiNum( m_moveDir,q_ddot, jntAcc);
END_METHOD

METHOD init : BOOL
VAR_INPUT
	i_startJntPos :Vec5d;
	i_targetJntPos :Vec5d;
	i_maxJntVel : Vec5d;
	i_maxJntAcc : Vec5d;
	i_maxJntJerk :Vec5d;
END_VAR
VAR 
	i:INT;
	maxV, maxA, maxJ :LREAL;
	q:ARRAY[1..2] OF LREAL;
	v:ARRAY[1..2] OF LREAL;
END_VAR
m_startPos:=i_startJntPos;
m_targetPos:=i_targetJntPos;
vecSub(i_targetJntPos, i_startJntPos, m_moveDir);
m_moveDistance := vecNorm(m_moveDir);

IF(m_moveDistance<g_smallNum) THEN
	vecMultiNum(g_onesVec7d,1/5, m_moveDir);;
ELSE
	vecMultiNum( m_moveDir,1/m_moveDistance, m_moveDir);
END_IF

// determian max vel/acc/jerk
maxV:=g_largeNum;
maxA:=g_largeNum;
maxJ:=g_largeNum;
FOR i :=1 TO 5 DO 
	IF ABS(m_moveDir[i])>g_smallNum THEN
		maxV := MIN (maxV, ABS(i_maxJntVel[i]/m_moveDir[i]));
		maxA := MIN (maxA, ABS(i_maxJntAcc[i]/m_moveDir[i]));
		maxJ := MIN (maxJ, ABS(i_maxJntJerk[i]/m_moveDir[i]));
	END_IF
END_FOR

// planning for moving distance
q[1]:=0;
q[2]:=m_moveDistance;
v[1]:=0;
v[2]:=0;
m_doubleS.init(q,v, maxV, maxA, maxJ);
m_duration:=m_doubleS.duration;
m_isGenerated:=m_doubleS.isGene;
END_METHOD

END_FUNCTION_BLOCK

// ---- Mains/RobotDynamics.TcPOU
PROGRAM RobotDynamics

VAR
	// slave robot arms joint data
	m_slaveJointsData AT %I* :ST_SlaveJointData;
	
	// setup joint5 position
	m_setupJointData AT %I* :ST_SetupJointData;
	
	// instrument info
	m_instruInfo AT %I* :ARRAY[1..g_sArmNum] OF ST_InstruStatus;
	
	// dynamic output
	m_slaveDynaData AT %Q* : ST_SlaveDynaData;
	m_setupJnt3Gravity AT %Q* : LREAL;
	m_setupJnt5Gravity AT %Q* : LREAL;
	
	// flag to init robot dynamic model
	m_robotDynaInit :BOOL :=FALSE;
	
	// grivity model block
	m_slaveGravityModel :ARRAY[1..g_sArmNum] OF FB_SlaveGravity;
	

	// code execute time measure
	m_codeTime : Profiler;
	
	// tmp variables
	i: INT;
	
END_VAR

m_codeTime(START:=TRUE, RESET:=TRUE);

// robot dynamic model init
IF m_robotDynaInit =FALSE THEN
	FOR i:=1 TO g_sArmNum DO
		m_slaveGravityModel[i].Init(i);
	END_FOR

	m_robotDynaInit:=TRUE;
END_IF

// run gravity model
FOR i:=1 TO g_sArmNum DO
	m_setupJointData.m_curJntPos[i][5]:=pi/2;
	m_slaveDynaData.m_gravity[i]:=m_slaveGravityModel[i].run(m_setupJointData.m_curJntPos[i][5], m_slaveJointsData.m_curJntPos[i],m_instruInfo[i]);

END_FOR

m_codeTime(START:=FALSE);

END_PROGRAM
